{attribute 'GeneratedUsingTerminal: EK1100-0000-0018'}
{attribute addProperty BoxType "EK1100-0000-0018"}
{attribute addProperty Id "Term_26_EL1819EL1819_32157CFD20Term_27_EL1819EL1819_32157CFD20Term_30_EL9011EL9011_D65D3D320"}
{attribute addProperty CRC "136412852"}
{attribute addProperty Size "40"}
{attribute addProperty Name "Term 25 (EK1100)"}
TYPE Term_25_EK1100_08217EB4 EXTENDS EK1100_1FC0878B :
STRUCT
	{attribute addProperty Name "Term 26 (EL1819)"}
	{attribute addProperty PreviousPort "Term 25 (EK1100) : B"}
	{attribute addProperty SyncUnit "Row_3"}
	Term_26_EL1819 : EL1819_32157CFD;
	{attribute addProperty Name "Term 27 (EL1819)"}
	{attribute addProperty PreviousPort "Term 26 (EL1819) : B"}
	{attribute addProperty SyncUnit "Row_3"}
	Term_27_EL1819 : EL1819_32157CFD;
	{attribute addProperty Name "Term 30 (EL9011)"}
	{attribute addProperty PreviousPort "Term 27 (EL1819) : B"}
	{attribute addProperty SyncUnit "default"}
	Term_30_EL9011 : EL9011_D65D3D32;
END_STRUCT
END_TYPE

(* stored: Version 1.2.0.0, ProductVersion 3.1.4024.11
   DUT Term_25_EK1100_08217EB4: Id {2975baa6-7d0d-4a67-bce3-f7bc8801b978} *)
